// TIA Portal project "Contatori" (V20)

(* hardware
DEVICE "S7-1200 station_1"  S7-1200 Station
   slot 0: "Rack_0"  S7-1200 Rack  Rack  V1.0
   slot 1: "Playground_PLC"  CPU 1214C DC/DC/DC  6ES7 214-1AG40-0XB0  V4.7
   slot 3: "AQ 1x12BIT_1"  AQ1 signal board  6ES7 232-4HA30-0XB0  V1.0
*)

// ===== PLC "Playground_PLC"  CPU 1214C DC/DC/DC =====

VAR_GLOBAL   // PLC tag table "Default tag table"
   "INPUT_CTU" AT %M0.0 : Bool;
   "INPUT_CTD" AT %M0.1 : Bool;
   "RESET_CTU" AT %M0.2 : Bool;
   "RESET_CTD" AT %M0.3 : Bool;
   "OUTPUT_CTU" AT %M0.4 : Bool;
   "OUTPUT_CTD" AT %M0.5 : Bool;
END_VAR

// folder: System blocks/Program resources

DATA_BLOCK "IEC_Counter_0_DB"   // DB1
{ S7_Optimized_Access := 'TRUE' }
AUTHOR : Simatic
FAMILY : IEC
NAME : CNTR
VERSION : 1.0
// stored: InstanceOfName IEC_COUNTER
"IEC_COUNTER"
BEGIN
END_DATA_BLOCK

DATA_BLOCK "IEC_Counter_0_DB_1"   // DB2
{ S7_Optimized_Access := 'TRUE' }
AUTHOR : Simatic
FAMILY : IEC
NAME : CNTR
VERSION : 1.0
// stored: InstanceOfName IEC_COUNTER
"IEC_COUNTER"
BEGIN
END_DATA_BLOCK

// folder: (top level)

ORGANIZATION_BLOCK "Main"   // OB1, LAD, ProgramCycle
TITLE = "Main Program Sweep (Cycle)"
{ S7_Optimized_Access := 'TRUE' }
VERSION : 0.1
   VAR_INPUT
      Initial_Call : Bool;   // Initial call of this OB
      Remanence : Bool;   // =True, if remanent data are available
   END_VAR
BEGIN

REGION Network 1
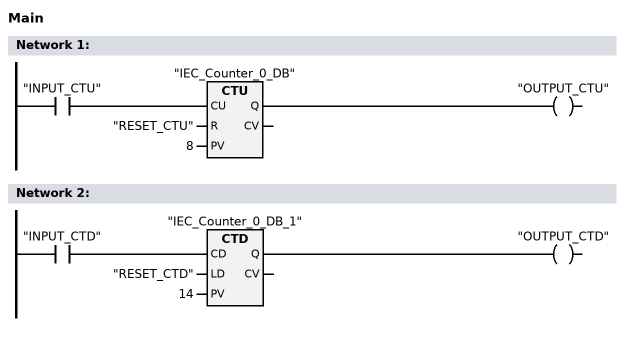
   "IEC_Counter_0_DB".CTU(CU := "INPUT_CTU", R := "RESET_CTU", PV := 8);
   "OUTPUT_CTU" := "IEC_Counter_0_DB".Q;
END_REGION

REGION Network 2
   "IEC_Counter_0_DB_1".CTD(CD := "INPUT_CTD", LD := "RESET_CTD", PV := 14);
   "OUTPUT_CTD" := "IEC_Counter_0_DB_1".Q;
END_REGION
END_ORGANIZATION_BLOCK